# EPICS IOC start-up script: test/startup/st.mcu035-twincat-ads.iocsh
epicsEnvSet("MOTOR_PORT",    "$(SM_MOTOR_PORT=MCU1)")
epicsEnvSet("IPADDR",        "$(SM_IPADDR=172.30.38.73)")
epicsEnvSet("IPPORT",        "$(SM_IPPORT=48898)")
epicsEnvSet("AMSNETIDIOC",   "$(SM_AMSNETID=172.30.38.12.1.1)")
epicsEnvSet("REMOTEAMSNETID", "5.36.136.2.1.1")
epicsEnvSet("ASYN_PORT",     "$(SM_ASYN_PORT=MC_CPU1)")
epicsEnvSet("SYSPFX",        "$(SM_SYSPFX=LabS-MCAG:MC-MCU-1035:)")
epicsEnvSet("P",             "$(SM_SYSPFX=LabS-MCAG:MC-MCU-1035:)")
epicsEnvSet("PREC",          "$(SM_PREC=3)")
epicsEnvSet("SM_NOAXES",     "1")
epicsEnvSet("ECM_OPTIONS",   "adsPort=852;amsNetIdRemote=$(REMOTEAMSNETID);amsNetIdLocal=$(AMSNETIDIOC)"

< ethercatmcController.iocsh

< ethercatmcEL6688-PTP-twincat-ads.iocsh

#####################################################
# EL1252, first channel TS_NS
epicsEnvSet("R",        "TS_NS")
epicsEnvSet("DESC",     "1Hz-TimeStamp ns")
epicsEnvSet("EGU",      "ns")
epicsEnvSet("ASYNADDR", "ADSPORT=852/GVL_APP.nTS_NS?")

< ethercatmcInt64in.iocsh
